(* CoDeSys 2.3 export: STDEVICESPACE.EXP *)

(* Data type *)
TYPE stDeviceSpace :
STRUCT
	byModbusSlaveAddress : BYTE;
	wModbusAdress : WORD;
	iModbusFunction : INT;
	pSPSDataSpace : DWORD;
	wSPSDataSpaceLength : WORD;
END_STRUCT
END_TYPE
